% RSLogix 500 project Practie-2.RSS, saved by version 8.30.00.16 %
PROJECT "UNTITLED"    % processor: MicroLogix 1000 %

PROGRAM FILES
  LAD 2 "MAIN_PROG"  4 rungs
  LAD 3 "USER_FAULT"  1 rungs
  LAD 4 "HSC_INT"  1 rungs
  LAD 5 "STI_INT"  1 rungs
  LAD 6, 7, 8, 9, 10, 11, 12, 13, 14, 15, 16: only END

DATA FILES
  O0 OUTPUT  1 elements
  I1 INPUT  2 elements
  S2 STATUS  33 elements
  B3 BINARY  32 elements
  T4 TIMER  40 elements
  C5 COUNTER  32 elements
  R6 CONTROL  16 elements
  N7 INTEGER  105 elements

LADDER 2 "MAIN_PROG"
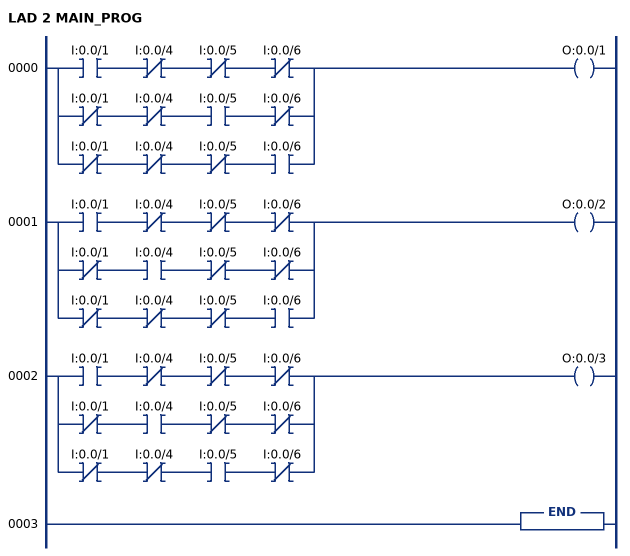
% Rung: 0 %
SOR BST XIC I:0.0/1 XIO I:0.0/4 XIO I:0.0/5 XIO I:0.0/6 NXB BST XIO I:0.0/1 XIO I:0.0/4 XIC I:0.0/5 XIO I:0.0/6 NXB XIO I:0.0/1 XIO I:0.0/4 XIO I:0.0/5 XIC I:0.0/6 BND BND OTE O:0.0/1 EOR
% Rung: 1 %
SOR BST XIC I:0.0/1 XIO I:0.0/4 XIO I:0.0/5 XIO I:0.0/6 NXB BST XIO I:0.0/1 XIC I:0.0/4 XIO I:0.0/5 XIO I:0.0/6 NXB XIO I:0.0/1 XIO I:0.0/4 XIO I:0.0/5 XIC I:0.0/6 BND BND OTE O:0.0/2 EOR
% Rung: 2 %
SOR BST XIC I:0.0/1 XIO I:0.0/4 XIO I:0.0/5 XIO I:0.0/6 NXB BST XIO I:0.0/1 XIC I:0.0/4 XIO I:0.0/5 XIO I:0.0/6 NXB XIO I:0.0/1 XIO I:0.0/4 XIC I:0.0/5 XIO I:0.0/6 BND BND OTE O:0.0/3 EOR
% Rung: 3 %
SOR END EOR
